PROGRAM Stn7ReturnPumpCtrl
VAR
END_VAR

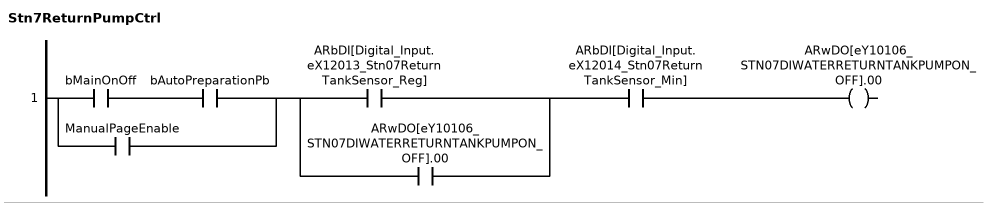
// NETWORK 1
ARwDO[eY10106_STN07DIWATERRETURNTANKPUMPON_OFF].00 := (bMainOnOff AND bAutoPreparationPb OR ManualPageEnable) AND (ARbDI[Digital_Input.eX12013_Stn07ReturnTankSensor_Reg] OR ARwDO[eY10106_STN07DIWATERRETURNTANKPUMPON_OFF].00) AND ARbDI[Digital_Input.eX12014_Stn07ReturnTankSensor_Min];

END_PROGRAM

(* stored: Version 1.1.0.1, ProductVersion 3.1.4024.12
   POU Stn7ReturnPumpCtrl: Id {8f6c9f7a-36e5-4e0f-840b-36e28f4fb394}, SpecialFunc None *)
